{attribute addProperty BoxType "EL3413-0000-0016"}
{attribute addProperty Id "PM_Inputs_ChannelAT %I*ARRAY[0..2] OF PM_Inputs_Channel_9FC8B9E8456570PM_Inputs_AuxiliaryAT %I*PM_Inputs_Auxiliary_4ACBD5CC6480PM_Outputs_ChannelAT %Q*ARRAY[0..2] OF PM_Outputs_Channel_A1108FBB2430PM_Outputs_AuxiliaryAT %Q*PM_Outputs_Auxiliary_4169B4F31620WcStateAT %I*WcState_F855686C1620InfoDataAT %I*InfoData_BC63D37F80100"}
{attribute addProperty CRC "4294487781"}
{attribute addProperty SizeInBites "656"}
{attribute addProperty SizeInBytes "82"}
TYPE EL3413_446C23E7 :
STRUCT
	{attribute addProperty Name "PM_Inputs_Channel"}
	PM_Inputs_Channel : ARRAY[0..2] OF PM_Inputs_Channel_9FC8B9E8;
	{attribute addProperty Name "PM_Inputs_Auxiliary"}
	PM_Inputs_Auxiliary : PM_Inputs_Auxiliary_4ACBD5CC;
	{attribute addProperty Name "PM_Outputs_Channel"}
	PM_Outputs_Channel : ARRAY[0..2] OF PM_Outputs_Channel_A1108FBB;
	{attribute addProperty Name "PM_Outputs_Auxiliary"}
	PM_Outputs_Auxiliary : PM_Outputs_Auxiliary_4169B4F3;
	{attribute addProperty Name "WcState"}
	WcState : WcState_F855686C;
	{attribute addProperty Name "InfoData"}
	InfoData : InfoData_BC63D37F;
END_STRUCT
END_TYPE

(* stored: Version 1.2.0.0, ProductVersion 3.1.4024.9
   DUT EL3413_446C23E7: Id {62b126d7-234c-449b-a6b4-771fa5efe25f} *)
